(* IEC 61131-3 sources: spire/plcs/jhu3, 1 file *)

(* ---- jhu3.st ---- *)
PROGRAM My_Program
  VAR
    transformer AT %QX0.0 : BOOL := 1;
    switch1 AT %QW0 : INT := 1;
    switch2 AT %QW1 : INT := 0;
    switch3 AT %QW2 : INT := 1;
    switch4 AT %QW3 : INT := 0;
    switch5 AT %QW4 : INT := 0;
    switch6 AT %QW5 : INT := 0;
  END_VAR

  switch6 := switch6;
END_PROGRAM

CONFIGURATION Config0

  RESOURCE Res0 ON PLC
    TASK TaskMain(INTERVAL := T#50ms,PRIORITY := 0);
    PROGRAM Inst0 WITH TaskMain : My_Program;
  END_RESOURCE
END_CONFIGURATION
